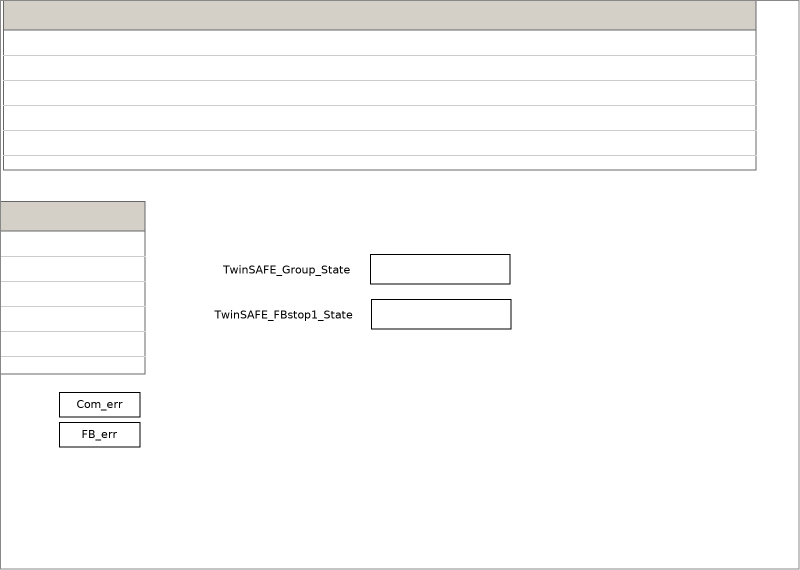
VISUALIZATION F99_IO_IO_1  // 800x570
    Table (3,0 753x170), data array: EL1904_M
        p3854506369: EL1904_M[1,INDEX]
        p1892666644: EL1904_M[2,INDEX]
        p338671338: EL1904_M[3,INDEX]
        p2170511999: EL1904_M[4,INDEX]
        p3723444502: EL1904_M[5,INDEX]
        Columns.Column.[0].Template: EL1904_M[1,INDEX]<>0
        Columns.Column.[1].Template: EL1904_M[2,INDEX]<>0
        Columns.Column.[2].Template: EL1904_M[3,INDEX]<>0
        Columns.Column.[3].Template: EL1904_M[4,INDEX]<>0
    Table (0,201 145x173), data array: EL2904
        p3854506369: EL2904[1,INDEX]
        p1892666644: EL2904[2,INDEX]
        p338671338: EL2904[3,INDEX]
        Columns.Column.[0].Template: EL2904[1,INDEX]<>0
    Rectangle (370,254 140x30), text list: 'TextList_TwinSAFE_Group_State', text index: P_TwinSAFE.TwinSAFE_Group_State
    Rectangle (371,299 140x30), text list: 'TextList_TwinSAFE_FB_ESTOP_State', text index: P_TwinSAFE.TwinSAFE_FBstop1_State
    Label (212,255 150x30), "TwinSAFE_Group_State"
    Label (209,300 150x30), "TwinSAFE_FBstop1_State"
    RoundedRectangle (59,422 81x25), "FB_err", colour toggle: P_TwinSAFE.FB_err
    RoundedRectangle (59,392 81x25), "Com_err", colour toggle: P_TwinSAFE.Com_err
END_VISUALIZATION

(* stored: Version 1.1.0.1, ProductVersion 3.1.4024.11
   Visu F99_IO_IO_1: Id {95475b4c-035b-4a78-9c6f-9e2613b65970} *)
